// tis is a class that is used by the ActorMovingTimeoutManager
TYPE ActorMovingTimeoutEx_t :
STRUCT
	ActorMovingTimeout : GernericErrorWatchdog_t;
	sensorPtr1 : POINTER TO BOOL := NULL;
	sensorPtr2 : POINTER TO BOOL := NULL;
	sensorPtr3 : POINTER TO BOOL := NULL;
	sensorID1 : sensorID_t := sensorID_t.SENSOR_NO_SENSOR;
	sensorID2 : sensorID_t := sensorID_t.SENSOR_NO_SENSOR;
	sensorID3 : sensorID_t := sensorID_t.SENSOR_NO_SENSOR;
END_STRUCT
END_TYPE

(* stored: Version 1.1.0.1
   DUT ActorMovingTimeoutEx_t: Id {c902e429-3e3d-4ba9-b54c-43f429a088b6} *)
